// SIMATIC S7-200 project (STEP 7-Micro/WIN), CPU 224 AM REL 19.07

ORGANIZATION_BLOCK 主程序:OB1
TITLE=程序注释
BEGIN
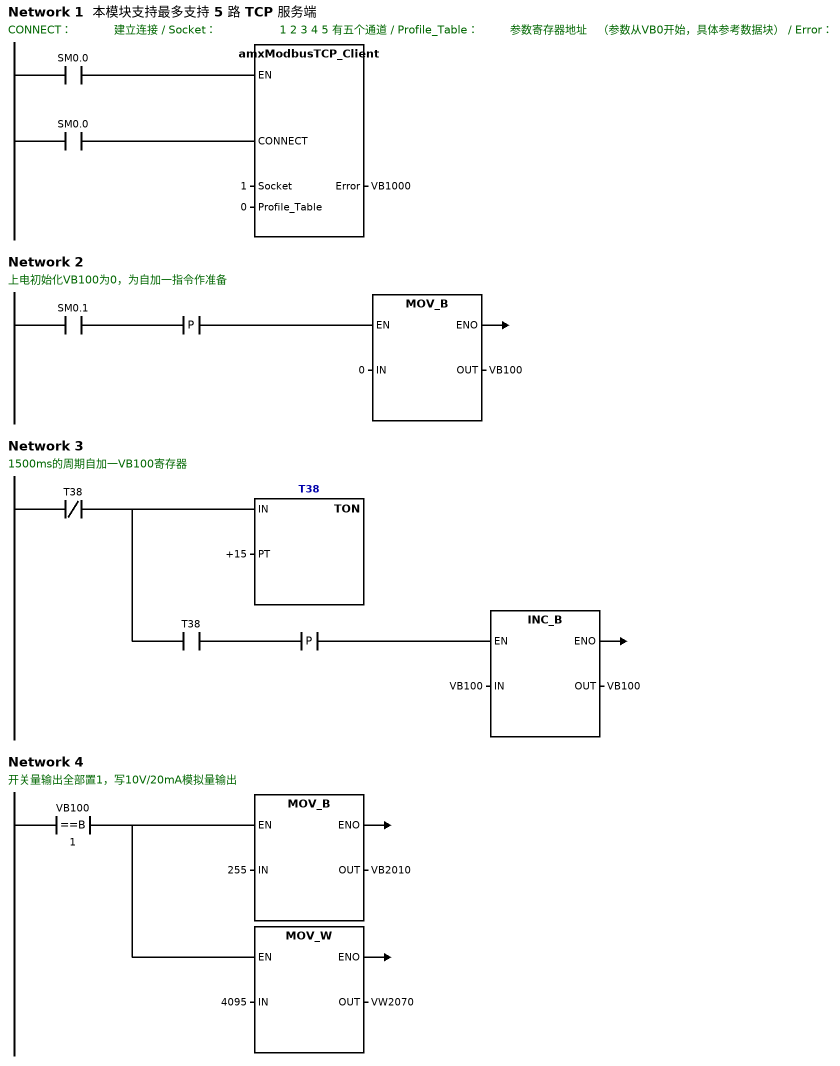
Network 1 // 本模块支持最多支持 5 路 TCP 服务端

// CONNECT：            建立连接
// Socket：                  1 2 3 4 5 有五个通道
// Profile_Table：         参数寄存器地址   （参数从VB0开始，具体参考数据块）
// Error：                      错误
LD     SM0.0
=      L60.0
LD     SM0.0
=      L63.7
LD     L60.0
CALL   amxModbusTCP_Client:SBR1, L63.7, 1, 0, VB1000
Network 2
// 上电初始化VB100为0，为自加一指令作准备
LD     SM0.1
EU
MOVB   0, VB100
Network 3
// 1500ms的周期自加一VB100寄存器
LDN    T38
TON    T38, +15
A      T38
EU
INCB   VB100
Network 4
// 开关量输出全部置1，写10V/20mA模拟量输出
LDB=   VB100, 1
MOVB   255, VB2010
MOVW   4095, VW2070
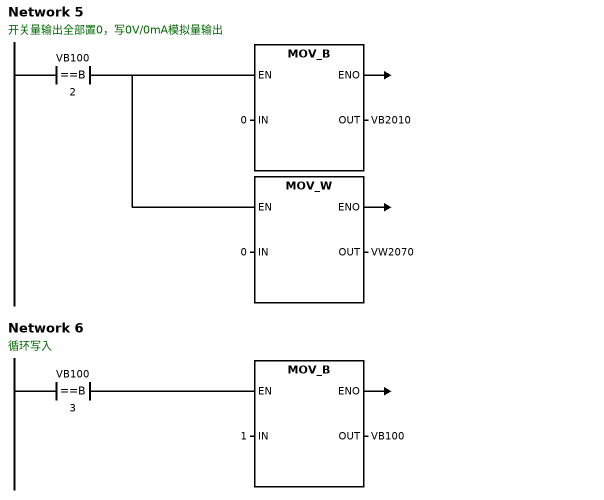
Network 5
// 开关量输出全部置0，写0V/0mA模拟量输出
LDB=   VB100, 2
MOVB   0, VB2010
MOVW   0, VW2070
Network 6
// 循环写入
LDB=   VB100, 3
MOVB   1, VB100
END_ORGANIZATION_BLOCK

// SBR1: protected block, not included

DATA_BLOCK_TAB 用户定义1
BEGIN
//通信口参数设置
VB0      4                   //本包络中包含的请求报文的段数                  
VB1      192                 //远端服务器的IP的最高字节
VB2      168                 //远端服务器的IP的第2字节
VB3      1                   //远端服务器的IP的第3字节
VB4      12                  //远端服务器的IP的第4字节
VB5      0                   //协议类型  0表示MODBUS TCP；1表示TCP传输
VB6      20                  //请求超时时间,单位：100MS
VW8      502                 //远端服务器的端口号
//第一段
VB10     1                   //从站站号
VB11     15                  //功能码 2读输入 1读线圈 5写单个线圈 15写多个线圈 4读输入寄存器 3读多个寄存器 6写单个寄存器 16写多个寄存器
VW14     1                   //读写MODBUS从站的数据地址  1线圈  10001输入  30001输入寄存器  40001保持寄存器
VW16     8                   //读写数据个数
VW18     2000                //V存贮器接收数据的起始地址  保存在VW2004开始的地址里
VW20     2010                //V存贮器发送数据的起始地址
//第二段
VB22     1                   //从站站号
VB23     2                   //功能码
VW26     10001               //读写MODBUS从站的数据地址
VW28     8                   //读写数据个数
VW30     2020                //V存贮器接收数据的起始地址（监控VB2024读IO8R模块8路开关量输入）
VW32     2030                //V存贮器发送数据的起始地址
//第三段
VB34     1                   //从站站号
VB35     4                   //功能码
VW38     30001               //读写MODBUS从站的数据地址
VW40     6                   //读写数据个数1
VW42     2040                //V存贮器接收数据的起始地址（监控VW2044~VW2049读IO模块6路模拟量输入值）
VW44     2050                //V存贮器发送数据的起始地址
//第四段
VB46     1                   //从站站号
VB47     6                   //功能码
VW50     40007               //读写MODBUS从站的数据地址
VW52     1                   //读写数据个数
VW54     2060                //V存贮器接收数据的起始地址
VW56     2070                //V存贮器发送数据的起始地址
END_DATA_BLOCK_TAB
